FUNCTION_BLOCK Drill (* Drill *)
  (* Standard: 61499-2 *)
  (* Version 0.2, 2003-12-04, JHC, Rockwell Automation, Renamed for better indexing. *)
  (* Version 0.1, 2002-11-05, JHC, Rockwell Automation, Corrected missing ST element in Algorithm REQ. *)
  (* Version 0.0, 2000-05-30, JHC, Rockwell Automation *)
  (* Compiler header: package fb.rt.benchmarks.DrillStation; *)
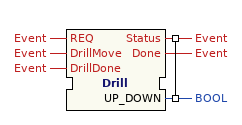
  EVENT_INPUT
    REQ; (* Normal Execution Request *)
    DrillMove; (* Simulate the time taken to move the drill *)
    DrillDone; (* Simulate the time taken to drill *)
  END_EVENT
  EVENT_OUTPUT
    Status WITH UP_DOWN;
    Done; (* Done drilling *)
  END_EVENT
  VAR_OUTPUT
    UP_DOWN : BOOL := true; (* true: up, false: down *)
  END_VAR
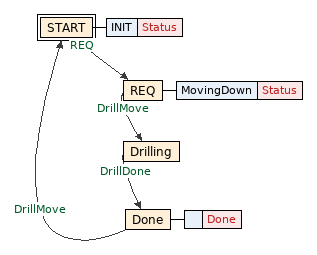
  EC_STATES
    START : INIT -> Status; (* Initial State *)
    REQ : MovingDown -> Status; (* Normal execution *)
    Done : -> Done;
    Drilling;
  END_STATES
  EC_TRANSITIONS
    START TO REQ := REQ;
    Done TO START := DrillMove;
    REQ TO Drilling := DrillMove;
    Drilling TO Done := DrillDone;
  END_TRANSITIONS
  ALGORITHM INIT IN ST: (* Initialization algorithm *)
UP_DOWN := TRUE;
  END_ALGORITHM
  ALGORITHM MovingDown IN ST: (* Normally executed algorithm *)
UP_DOWN := FALSE;
  END_ALGORITHM
END_FUNCTION_BLOCK
